// Mitsubishi GX Works2 project: LRI - Exercìcio 5   PLC: Q03UDV
// HelloWorld

PROGRAM MAIN
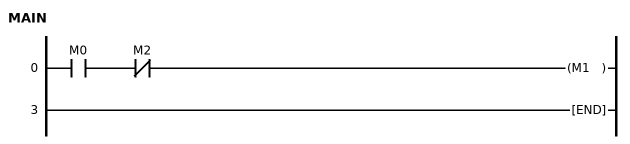
0     LD      M0
      ANI     M2
      OUT     M1
3     END
END_PROGRAM
